FUNCTION_BLOCK ABSTRACT SmartHome
VAR_GENERIC CONSTANT
    _DeviceCount : UDINT := 1;
END_VAR
VAR_OUTPUT
	Devices : ARRAY [0.._DeviceCount - 1] OF IDevice;
END_VAR
VAR
	_SavedDeviceStates : ARRAY [0.._DeviceCount - 1] OF DEVICE_STATE;
	
	_LogMessageCounter : UDINT;
END_VAR

METHOD Execute
updateInputDevices();

OnTick();

updateOutputDevices();

saveDevicesState();
END_METHOD

//FB_Init is always available implicitly and it is used primarily for initialization.
//The return value is not evaluated. For a specific influence, you can also declare the
//methods explicitly and provide additional code there with the standard initialization
//code. You can evaluate the return value.
METHOD FB_Init: BOOL
VAR_INPUT
    bInitRetains: BOOL; // TRUE: the retain variables are initialized (reset warm / reset cold)
    bInCopyCode: BOOL;  // TRUE: the instance will be copied to the copy code afterward (online change)   
END_VAR
Devices := GetDeviceArray();
END_METHOD

METHOD PROTECTED ABSTRACT GetDeviceArray : ARRAY [0.._DeviceCount - 1] OF IDevice
END_METHOD

METHOD PRIVATE logDevicesState
VAR
	i : UDINT;
	message : STRING;
END_VAR
FOR i := 0 TO _DeviceCount - 1 DO
	IF Devices[i].State = DEVICE_STATE.FAULT AND_THEN _SavedDeviceStates[i] <> DEVICE_STATE.FAULT THEN
		_LogMessageCounter := _LogMessageCounter + 1;
		
		message := Tc2_Standard.CONCAT(
			Tc2_Standard.CONCAT(
				Tc2_Standard.CONCAT('#', TO_STRING(_LogMessageCounter)),
				Tc2_Standard.CONCAT(': ', 'Device "')
			),
			Tc2_Standard.CONCAT(
				Tc2_Standard.CONCAT(Devices[i].Name, '" at "'),
				Tc2_Standard.CONCAT(Devices[i].Place, '" is in fault state')
			)
		);
			
		Tc2_System.ADSLOGSTR(msgCtrlMask := Tc2_System.Global_Variables.ADSLOG_MSGTYPE_ERROR, message, '');
	ELSIF Devices[i].State = DEVICE_STATE.WORKING AND_THEN _SavedDeviceStates[i] <> DEVICE_STATE.WORKING THEN
		_LogMessageCounter := _LogMessageCounter + 1;

		message := Tc2_Standard.CONCAT(
			Tc2_Standard.CONCAT(
				Tc2_Standard.CONCAT('#', TO_STRING(_LogMessageCounter)),
				Tc2_Standard.CONCAT(': ', 'Device "')
			),
			Tc2_Standard.CONCAT(
				Tc2_Standard.CONCAT(Devices[i].Name, '" at "'),
				Tc2_Standard.CONCAT(Devices[i].Place, '" is in working state')
			)
		);
			
		Tc2_System.ADSLOGSTR(msgCtrlMask := Tc2_System.Global_Variables.ADSLOG_MSGTYPE_HINT, message, '');		
	END_IF
END_FOR
END_METHOD

METHOD PROTECTED OnTick
logDevicesState();
END_METHOD

METHOD PRIVATE saveDevicesState
VAR
	i : UDINT;
END_VAR
FOR i := 0 TO _DeviceCount - 1 DO
	_SavedDeviceStates[i] := Devices[i].State;
END_FOR
END_METHOD

METHOD PRIVATE updateInputDevices
VAR
	i : UDINT;
	device : IDevice;
	inputDevice : IInputDevice;
END_VAR
FOR i := 0 TO _DeviceCount - 1 DO
	device := Devices[i];
	
	IF __QUERYINTERFACE(device, inputDevice) THEN
		inputDevice.ReadInputs();		
	END_IF
END_FOR
END_METHOD

METHOD PRIVATE updateOutputDevices
VAR
	i : UDINT;
	device : IDevice;
	outputDevice : IOutputDevice;
END_VAR
FOR i := 0 TO _DeviceCount - 1 DO
	device := Devices[i];
	
	IF __QUERYINTERFACE(device, outputDevice) THEN
		outputDevice.WriteOutputs();		
	END_IF
END_FOR
END_METHOD

END_FUNCTION_BLOCK

(* stored: Version 1.1.0.1
   POU SmartHome: Id {857a971e-5d7c-4106-8e02-185b2c21ea0c}, SpecialFunc None
   Folder Members to override: Id {76ab9287-c394-47e6-a14d-89ef40e1a3ee}
   Folder Private members: Id {f591475b-63c4-45e9-b3b9-ccf9d984630b}
   Method Execute: Id {9c1a966d-9ec6-43cd-a154-c4059e37e7a5}
   Method FB_Init: Id {3e5e8d01-45db-4578-be3e-4146897eccb5}
   Method GetDeviceArray: Id {46d5259b-25e6-40bc-bda7-1ffa1812e176}
   Method logDevicesState: Id {b46d7961-31c0-4d73-8d43-3b3a197424ca}
   Method OnTick: Id {c3d4dc74-548b-46fb-9af8-1188cc74d0a6}
   Method saveDevicesState: Id {c2735e41-08c5-48a6-bc0c-ffc69f2f81c2}
   Method updateInputDevices: Id {f46dab79-235e-415c-a629-ad81b71c0555}
   Method updateOutputDevices: Id {07929116-9320-4b69-87e5-3c210c3fa6f1} *)
